// TIA Portal V16 export
// export: Created 2024-09-05T17:39:15.9150643Z, ExportSetting WithDefaults, DisplayName Totally Integrated Automation Portal, DisplayVersion V16 Update 6, DisplayName TIA Portal Version Control Interface, DisplayVersion V16 Update 2, DisplayName TIA Portal Openness, DisplayVersion V16 Update 6, DisplayName STEP 7 Professional, DisplayVersion V16 Update 6, DisplayName STEP 7 Safety, DisplayVersion V16, DisplayName WinCC Advanced, DisplayVersion V16 Update 6
ORGANIZATION_BLOCK "OB_RackStationFailure"   // OB86, LAD, RackOrStationFailure
{ S7_Optimized_Access := 'TRUE' }
VERSION : 0.1
// stored: IsIECCheckEnabled false, SetENOAutomatically false
   VAR_INPUT
      LADDR : HW_DEVICE;   // Hardware identifier
      Event_Class : Byte;   // Event class
      Fault_ID : Byte;   // Fault identifier
   END_VAR
BEGIN
END_ORGANIZATION_BLOCK
